TYPE typeEtherCATState :
STRUCT
	//suffix code
	//0x___1 = Slave in 'INIT' state
	//0x___2 = Slave in 'PREOP' state
	//0x___3 = Slave in 'BOOT' state
	//0x___4 = Slave in 'SAFEOP' state
	//0x___8 = Slave in 'OP' state
	state:EtherCATstate;

	
	
	//prefix code
	//0x001_ = Slave signals error
	//0x002_ = Invalid vendorId, productCode... read
	//0x004_ = Initialization error occurred
	//0x008_ = Slave disabled
	//0x010_ = Slave not present
	//0x020_ = Slave signals link error
	//0x040_ = Slave signals missing link
	//0x080_ = Slave signals unexpected link
	//0x100_ = Communication port A
	//0x200_ = Communication port B
	//0x400_ = Communication port C
	//0x800_ = Communication port D
	suffix:EtherCATSuffix;
	
	isFault:BOOL; //TRUE if either state is not 8 and code exists
	colour:DWORD; //colour state
	
	

END_STRUCT
END_TYPE

(* stored: Version 1.1.0.1, ProductVersion 3.1.4024.12
   DUT typeEtherCATState: Id {664d9b35-bbb5-48a5-8c1a-cacd73768969} *)
